// TIA Portal V18 export
// export: Created 2026-03-12T16:04:35.124399Z, ExportSetting WithDefaults, DisplayName Totally Integrated Automation Portal, DisplayVersion V18 Update 5, DisplayName TIA Portal Openness, DisplayVersion V18 Update 5, DisplayName TIA Portal Version Control Interface, DisplayVersion V18, DisplayName SINAMICS Startdrive Advanced, DisplayVersion V18, DisplayName SINAMICS Startdrive G130, G150, S120, S150, SINAMICS MV, S210, DisplayVersion V18, DisplayName SINAMICS Startdrive G110M, G120, G120C, G120D, G120P, G115D, DisplayVersion V18, DisplayName STEP 7 Professional, DisplayVersion V18 Update 5, DisplayName STEP 7 Safety, DisplayVersion V18, DisplayName WinCC Professional, DisplayVersion V18 Update 5
FUNCTION_BLOCK "FB STATUS MOTOR"   // FB35, LAD
{ S7_Optimized_Access := 'TRUE' }
VERSION : 0.1
// stored: AutoNumber true, IsIECCheckEnabled false, IsRetainMemResEnabled false, MemoryReserve 100, SetENOAutomatically false, UDAEnableTagReadback false
   VAR_INPUT
      INPUT_LIGADO : Bool;   // 1 = Sinal elétrico de campo indicando bomba ligada
      INPUT_FALHA : Bool;   // 0 = Sinal elétrico de campo indicando bomba em falha
      FALHA_COMUNICACAO : Bool;
   END_VAR
   VAR_OUTPUT
      STATUS_MOTOR : Byte;   // 0 = DESLIGADO; 1 = LIGADO; 2 = FALHA; 3 = MANUTENÇÃO; 4 = SEM COMUNICAÇÃO MODBUS
   END_VAR
BEGIN

REGION Network 1: Recebimento dos sinais de entrada (Sinais de campo e comandos)
   // INPUT_ABERTA = Entrada de sinal de Bomba Ligada
   // INPUT_FECHADA = Entrada de sinal de Bomba Desligada
   // INPUT_FALHA = Entrada de sinal de Bomba em Falha
   // INPUT_FALHA_PROFINET = Sem comunicação Profinet
   // STATUS_MOTOR: 0 = DESLIGADO; 1 = LIGADO; 2 = FALHA; 3 = MANUTENÇÃO; 4 = SEM COMUNICAÇÃO MODBUS
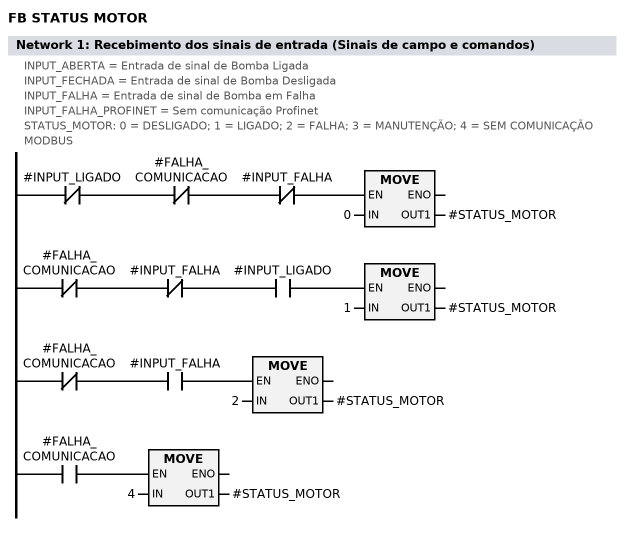
   RUNG wire#powerrail
      I_Contact( #INPUT_LIGADO )
      I_Contact( #FALHA_COMUNICACAO )
      I_Contact( #INPUT_FALHA )
      Move(in := 0, out1 => #STATUS_MOTOR)
   END_RUNG
   RUNG wire#powerrail
      I_Contact( #FALHA_COMUNICACAO )
      I_Contact( #INPUT_FALHA )
      Contact( #INPUT_LIGADO )
      Move(in := 1, out1 => #STATUS_MOTOR)
   END_RUNG
   RUNG wire#powerrail
      I_Contact( #FALHA_COMUNICACAO )
      Contact( #INPUT_FALHA )
      Move(in := 2, out1 => #STATUS_MOTOR)
   END_RUNG
   RUNG wire#powerrail
      Contact( #FALHA_COMUNICACAO )
      Move(in := 4, out1 => #STATUS_MOTOR)
   END_RUNG
   // the same network as SCL:
   IF NOT #INPUT_LIGADO AND NOT #FALHA_COMUNICACAO AND NOT #INPUT_FALHA THEN #STATUS_MOTOR := 0; END_IF;
   IF NOT #FALHA_COMUNICACAO AND NOT #INPUT_FALHA AND #INPUT_LIGADO THEN #STATUS_MOTOR := 1; END_IF;
   IF NOT #FALHA_COMUNICACAO AND #INPUT_FALHA THEN #STATUS_MOTOR := 2; END_IF;
   IF #FALHA_COMUNICACAO THEN #STATUS_MOTOR := 4; END_IF;
END_REGION
END_FUNCTION_BLOCK
